SUBAPPLICATION mapping_aux (* Subapplication Type *)
  (* Standard: 61499-2 *)
  (* Version 1.0, 2023-01-29, Franz *)
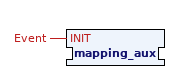
  EVENT_INPUT
    INIT;
  END_EVENT
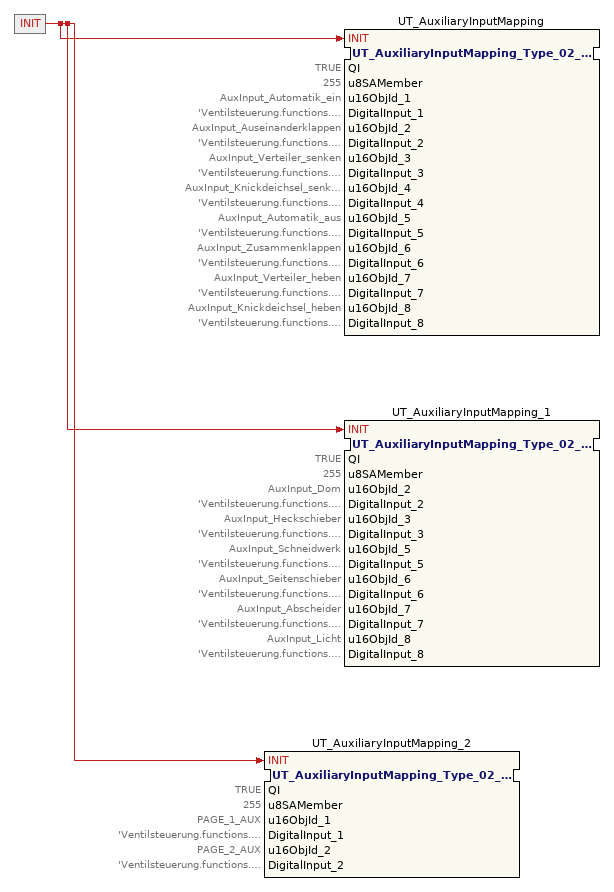
  FBS
    UT_AuxiliaryInputMapping : UT_AuxiliaryInputMapping_Type_02_Bool_NonLatched(QI := TRUE, u8SAMember := 255, u16ObjId_1 := AuxInput_Automatik_ein, DigitalInput_1 := 'Ventilsteuerung.functions.Automatik.ein.AuxInput', u16ObjId_2 := AuxInput_Auseinanderklappen, DigitalInput_2 := 'Ventilsteuerung.functions.Klappen.AuxInput_heben.IX', u16ObjId_3 := AuxInput_Verteiler_senken, DigitalInput_3 := 'Ventilsteuerung.functions.Verteiler.AuxInput_senken.IX', u16ObjId_4 := AuxInput_Knickdeichsel_senken, DigitalInput_4 := 'Ventilsteuerung.functions.Knickdeichsel.AuxInput_senken.IX', u16ObjId_5 := AuxInput_Automatik_aus, DigitalInput_5 := 'Ventilsteuerung.functions.Automatik.aus.AuxInput', u16ObjId_6 := AuxInput_Zusammenklappen, DigitalInput_6 := 'Ventilsteuerung.functions.Klappen.AuxInput_senken.IX', u16ObjId_7 := AuxInput_Verteiler_heben, DigitalInput_7 := 'Ventilsteuerung.functions.Verteiler.AuxInput_heben.IX', u16ObjId_8 := AuxInput_Knickdeichsel_heben, DigitalInput_8 := 'Ventilsteuerung.functions.Knickdeichsel.AuxInput_heben.IX');
    UT_AuxiliaryInputMapping_1 : UT_AuxiliaryInputMapping_Type_02_Bool_NonLatched(QI := TRUE, u8SAMember := 255, u16ObjId_2 := AuxInput_Dom, DigitalInput_2 := 'Ventilsteuerung.functions.Dom.AuxInput_UP.IX', u16ObjId_3 := AuxInput_Heckschieber, DigitalInput_3 := 'Ventilsteuerung.functions.Heckschieber.AuxInput_UP.IX', u16ObjId_5 := AuxInput_Schneidwerk, DigitalInput_5 := 'Ventilsteuerung.functions.Schneidwerk.AuxInput_UP.IX', u16ObjId_6 := AuxInput_Seitenschieber, DigitalInput_6 := 'Ventilsteuerung.functions.Seitenschieber.AuxInput_UP.IX', u16ObjId_7 := AuxInput_Abscheider, DigitalInput_7 := 'Ventilsteuerung.functions.Abscheider.AuxInput_UP.IX', u16ObjId_8 := AuxInput_Licht, DigitalInput_8 := 'Ventilsteuerung.functions.Licht.AuxInput_UP.IX');
    UT_AuxiliaryInputMapping_2 : UT_AuxiliaryInputMapping_Type_02_Bool_NonLatched(QI := TRUE, u8SAMember := 255, u16ObjId_1 := PAGE_1_AUX, DigitalInput_1 := 'Ventilsteuerung.functions.PAGES.PAGE_1.AUX', u16ObjId_2 := PAGE_2_AUX, DigitalInput_2 := 'Ventilsteuerung.functions.PAGES.PAGE_2.AUX');
  END_FBS
  EVENT_CONNECTIONS
    INIT TO UT_AuxiliaryInputMapping.INIT;
    INIT TO UT_AuxiliaryInputMapping_1.INIT;
    INIT TO UT_AuxiliaryInputMapping_2.INIT;
  END_CONNECTIONS
END_SUBAPPLICATION
